FUNCTION Convert_ULINT_TO_INT : Hresult
VAR_INPUT
	in : ULINT;
	out : REFERENCE TO INT;
END_VAR
VAR
	converted : INT;
END_VAR
VAR CONSTANT
	INCOMPATIBLE : HRESULT := 16#9811070E;
END_VAR

converted := ULINT_TO_INT(in);

IF (INT_TO_ULINT(converted) <> in) THEN
	Convert_ULINT_TO_INT := INCOMPATIBLE;
	RETURN;
END_IF

out := converted;

END_FUNCTION

(* stored: Version 1.1.0.1, ProductVersion 3.1.4024.12
   POU Convert_ULINT_TO_INT: Id {e4c75813-1b67-4dcf-b674-7f801bec62e4}, SpecialFunc None *)
